Omron CX-Programmer project NewProject (CX-Programmer 9.61)

# PLC NewPLC1: CJ1M CPU22
I/O table (CPU CJ1M-CPU22): rack 0 slot 0 CJ1W-ID211; rack 0 slot 1 CJ1W-OC211; rack 0 slot 2 CJ1W-MAD42

## Global symbols (name address type ; comment)
0.00 BOOL  ; start
0.01 BOOL  ; stop
0.02 BOOL  ; regulersize
0.03 BOOL  ; bigsize
0.04 BOOL  ; p1
0.05 BOOL  ; p2
1.00 BOOL  ; con1
1.01 BOOL  ; con2
1.02 BOOL  ; selenoid
1.03 BOOL  ; run
1.04 BOOL  ; setRegulerSize
1.05 BOOL  ; setBigSize
3 CHANNEL  ; P1
C0000 BOOL  ; count_P1
C0001 BOOL  ; count_P2
T0000 BOOL  ; T_regulerSize
T0001 BOOL  ; T_bigSize
W0.00 BOOL  ; start
W0.01 BOOL  ; stop
W0.02 BOOL  ; regulerSize
W0.03 BOOL  ; bigSize
W0.04 BOOL  ; P1
W0.06 BOOL  ; run
W0.07 BOOL  ; setRegulerSize
W0.08 BOOL  ; setBigSize

## Program NewProgram1 (cyclic task 0)
Local symbols
t BOOL

### Section Section1

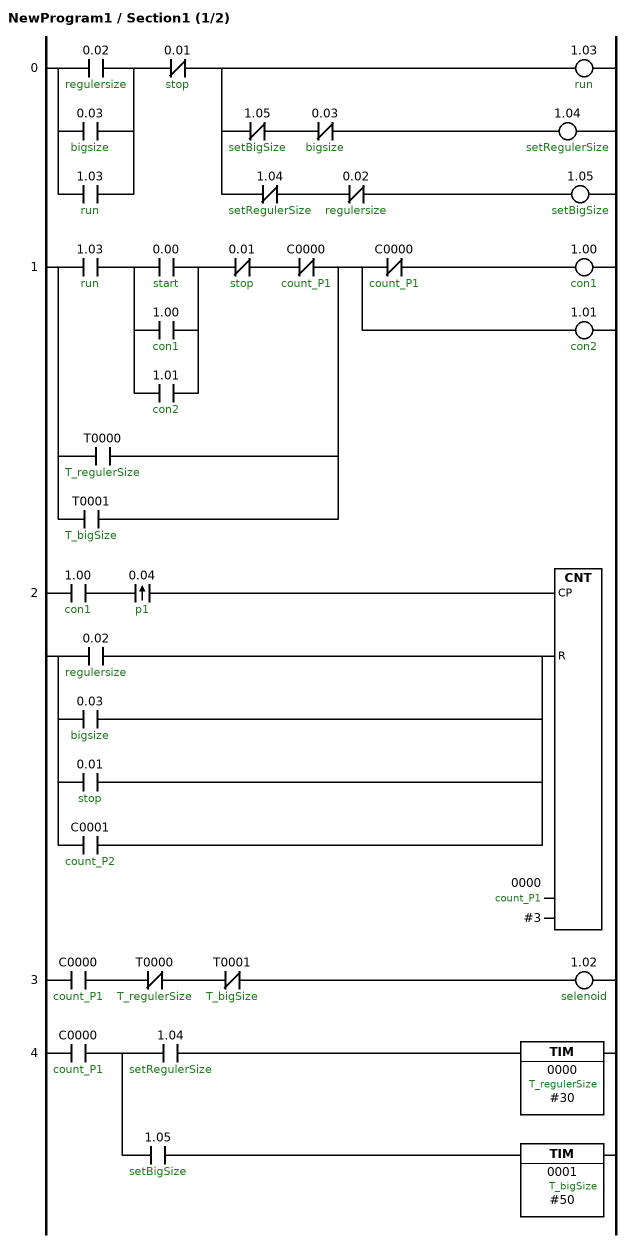
; rung 0
LD 0.02  ; regulersize
OR 0.03  ; bigsize
OR 1.03  ; run
ANDNOT 0.01  ; stop
OUT TR0
OUT 1.03  ; run
ANDNOT 1.05  ; setBigSize
ANDNOT 0.03  ; bigsize
OUT 1.04  ; setRegulerSize
LD TR0
ANDNOT 1.04  ; setRegulerSize
ANDNOT 0.02  ; regulersize
OUT 1.05  ; setBigSize
; rung 1
LD 1.03  ; run
LD 0.00  ; start
OR 1.00  ; con1
OR 1.01  ; con2
ANDLD
ANDNOT 0.01  ; stop
ANDNOT C0000  ; count_P1
OR T0000  ; T_regulerSize
OR T0001  ; T_bigSize
OUT TR0
ANDNOT C0000  ; count_P1
OUT 1.00  ; con1
LD TR0
OUT 1.01  ; con2
; rung 2
LD 1.00  ; con1
@AND 0.04  ; p1
LD 0.02  ; regulersize
OR 0.03  ; bigsize
OR 0.01  ; stop
OR C0001  ; count_P2
CNT 0000 #3  ; count_P1
; rung 3
LD C0000  ; count_P1
ANDNOT T0000  ; T_regulerSize
ANDNOT T0001  ; T_bigSize
OUT 1.02  ; selenoid
; rung 4
LD C0000  ; count_P1
OUT TR0
AND 1.04  ; setRegulerSize
TIM 0000 #30  ; T_regulerSize
LD TR0
AND 1.05  ; setBigSize
TIM 0001 #50  ; T_bigSize

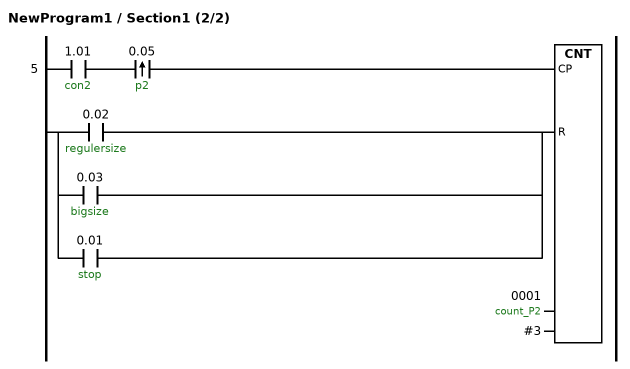
; rung 5
LD 1.01  ; con2
@AND 0.05  ; p2
LD 0.02  ; regulersize
OR 0.03  ; bigsize
OR 0.01  ; stop
CNT 0001 #3  ; count_P2

### Section END
; rung 0
END(001)